// TIA Portal V17 export
// export: Created 2026-04-13T11:12:04.3157831Z, ExportSetting WithDefaults, DisplayName Totally Integrated Automation Portal, DisplayVersion V17 Update 4, DisplayName TIA Portal Openness, DisplayVersion V17 Update 4, DisplayName TIA Portal Version Control Interface, DisplayVersion V17, DisplayName SINAMICS Startdrive Advanced, DisplayVersion V17, DisplayName SINAMICS Startdrive G130, G150, S120, S150, SINAMICS MV, S210, DisplayVersion V17, DisplayName SINAMICS Startdrive G110M, G120, G120C, G120D, G120P, G115D, DisplayVersion V17, DisplayName STEP 7 Professional, DisplayVersion V17 Update 4, DisplayName STEP 7 Safety, DisplayVersion V17, DisplayName WinCC Professional, DisplayVersion V17 Update 4
DATA_BLOCK "BY2"   // DB24
{ S7_Optimized_Access := 'TRUE' }
VERSION : 0.1
// stored: AutoNumber true, DBAccessibleFromOPCUA true, DBAccessibleFromWebserver true, IsOnlyStoredInLoadMemory false, IsRetainMemResEnabled false, IsWriteProtectedInAS false, MemoryReserve 100
   VAR
      MBY等待保压 : Bool;
      MBY正在充气 : Bool;
      MBY保压不佳 : Bool;
      MBY正在保压 : Bool;
      MBY保压正常 : Bool;
      MBY保压 : Bool;
      MQT其他阀 : Bool;
      MCQ充气阀 : Bool;
      当前阶段 : Int;
   END_VAR
   VAR RETAIN
      SV低设定 : Real;
      SV高设定 : Real;
      SV保压差值 : Real;
      SV保压时 : UInt;
      SV保压分 : UInt;
      SV保压秒 : UInt;
   END_VAR
   VAR
      PV塔内压力 : Real;
      PV保压前 : Real;
      PV保压后 : Real;
      PV当前差值 : Real;
      PV保压时 : UInt;
      PV保压分 : UInt;
      PV保压秒 : UInt;
   END_VAR
BEGIN
END_DATA_BLOCK
